(* CoDeSys 2.3 export: FK14PUMPSFAULTYCONTROL.EXP *)

(* POU K14/fK14PumpsFaultyControl, ST *)
FUNCTION fK14PumpsFaultyControl : BOOL
(* Проверка состояния насосов*)
VAR_INPUT
	PumpState : ARRAY [1..MAX_K14_PUMPS_NUM] OF BOOL;
	PumpStatusCheckDelay : ARRAY [1..MAX_K14_PUMPS_NUM] OF BOOL;
	PressureDrop : BOOL;
END_VAR
VAR
	i : USINT;
	activePumpID : USINT; (*номер работающего насоса*)
END_VAR
activePumpID := 0;

FOR i := 1 TO MAX_K14_PUMPS_NUM DO
	IF PumpState[i] THEN
		IF activePumpID <> 0 THEN
			(*
				Включено больше одного насоса -
				ничего не можем сказать об их исправности
			*)
			RETURN;
		END_IF;
		activePumpID := i;
	END_IF;
END_FOR;

IF activePumpID = 0 THEN
	(*
		Не включен ни один насос - 
		ничего не можем сказать об их исправности
	*)
	RETURN;
END_IF;

IF PumpStatusCheckDelay[activePumpID] THEN
	(*
		Определяем исправность насоса
		по перепаду давления
	*)
	K14PumpFaulty[activePumpID] := NOT(PressureDrop);
END_IF;
END_FUNCTION
